Universal Robots PolyScope program: d_to_c.urp

Program d_to_c (installation=string_planes directory=/programs/string_crossings createdIn=5.17.3 lastSavedIn=5.17.3 robotSerialNumber=20245501435)
Calibrated DH parameters: a=[0.000154, -0.137004, -0.385524, -0.00002, 0.000092, 0]; d=[0.162441, 211.794786, -230.585024, 18.923638, 0.099786, 0.09951]; alpha=[1.569493, -0.001902, 0.003874, 1.570111, -1.570167, 0]; deltaTheta=[0, -1.242934, 1.056292, 0.186646, 0.000002, 0.000001]
InitVariablesNode
Robot Program (runOnlyOnce=false)
  bow_section := -1
  If bow_section≟-1
    MoveJ speed 60 deg/s, acceleration 80 deg/s^2 (useActiveTCP=true) feature=Base
      Waypoint Waypoint_2 (Relative): relativeFromPosition TCP in base x=316.087 y=723.603 z=117.786 mm, rx=-1.5349 ry=-2.2386 rz=1.1275 rad; joints [-128.46, -21.869, 50.823, -72.931, -81.954, -152.853] deg; TCP offset x=28.21 y=-96.107 z=-99.69 mm, rx=0 ry=0 rz=0 rad; TCP in base x=245.285 y=570.708 z=53.285 mm, rx=-1.8425 ry=-1.3918 rz=0.0687 rad; joints [-132.226, -24.799, 96.314, -169.323, -42.691, -112.607] deg
  ElseIf bow_section≟0
    MoveJ speed 60 deg/s, acceleration 80 deg/s^2 (useActiveTCP=true) feature=Base
      Waypoint Waypoint_1 (Relative): relativeFromPosition TCP in base x=337.283 y=452.564 z=146.255 mm, rx=-1.6083 ry=-2.1978 rz=1.0429 rad; joints [-146.229, -47.167, 100.75, -99.804, -91.441, -163.026] deg; TCP in base x=195.29 y=411.468 z=21.275 mm, rx=-1.7343 ry=-1.5169 rz=0.4321 rad; joints [-140.233, -30.937, 122.531, -154.99, -45.8, -143.197] deg
  Else 
    MoveJ speed 60 deg/s, acceleration 80 deg/s^2 (useActiveTCP=true) feature=Base
      Waypoint Waypoint_3 (Relative): relativeFromPosition TCP in base x=340.787 y=238.628 z=127.316 mm, rx=-1.5374 ry=-2.1222 rz=1.0864 rad; joints [-167.853, -53.466, 123.57, -113.68, -104.543, -179.467] deg; TCP in base x=152.628 y=275.821 z=-5.995 mm, rx=-1.6121 ry=-1.6008 rz=0.7404 rad; joints [-153.501, -26.651, 138.52, -151.349, -62.642, -165.796] deg
